FUNCTION_BLOCK FB_ScopeServer
VAR_INPUT
	//sNetId					: STRING	:='';	
    bExternalTriggerEvent	: BOOL 	:= FALSE; //Rising edge start recording, falling edge stop and save
	sConfigFile				: STRING; //.tcscopex
	sSaveFile				: STRING; //.svdx
END_VAR
//VAR_OUTPUT
VAR
    bBusy					: BOOL 		:= FALSE;
    bError					: BOOL 		:= FALSE;
    nErrorId				: UDINT 	:= 0;	
END_VAR
VAR

    bDone					: BOOL 		:= FALSE;	

    fbScopeServerControl	: FB_ScopeServerControl;
    eReqState				: E_ScopeServerState := SCOPE_SERVER_IDLE;
	
    eState					: (IDLE,RECORDING,SAVING,DISCONNECTING,ERROR,RESETING);
END_VAR

CASE eState OF
	IDLE:
		bBusy	:=FALSE;
		IF bExternalTriggerEvent THEN
			bBusy			:= TRUE;
	    	eReqState 		:= SCOPE_SERVER_START;
	    	eState 			:= RECORDING;	
		END_IF
	
	RECORDING:	
		IF fbScopeServerControl.bDone THEN
	    	IF NOT bExternalTriggerEvent THEN
	    	    eReqState 		:= SCOPE_SERVER_SAVE;
	    	    eState 			:= SAVING;
	    	END_IF
		ELSIF fbScopeServerControl.bError THEN
			eState	:=ERROR;		
		END_IF
		
	SAVING:
	    IF fbScopeServerControl.bDone THEN
	        eReqState 		:= SCOPE_SERVER_DISCONNECT;
			eState			:= DISCONNECTING;
		ELSIF fbScopeServerControl.bError THEN
			eState	:=ERROR;		
		END_IF
		
	DISCONNECTING:
		IF fbScopeServerControl.bDone THEN
	       eState := IDLE;
		ELSIF fbScopeServerControl.bError THEN
			eState	:=ERROR;				   
	    END_IF		
		
	ERROR:
		bBusy			:= FALSE;
		IF NOT bExternalTriggerEvent THEN
			bBusy			:= TRUE;
			eReqState 		:= SCOPE_SERVER_RESET;
			eState			:= DISCONNECTING;
		END_IF
		
	RESETING:
		IF fbScopeServerControl.bDone OR fbScopeServerControl.bError THEN
	       	eReqState 		:= SCOPE_SERVER_IDLE;
			eState			:= IDLE; 
	    END_IF		
		
END_CASE


fbScopeServerControl( sNetId		:= '',
                      eReqState		:= eReqState,
                      sConfigFile	:= sConfigFile,
                      sSaveFile		:= sSaveFile,
                      tTimeout		:= T#10S,
                      bBusy			=>,
                      bDone			=>bDone,
                      bError		=>bError,
                      nErrorId		=>nErrorId);

END_FUNCTION_BLOCK

(* stored: Version 1.1.0.1
   POU FB_ScopeServer: Id {2a934d08-2426-4f56-8017-5dfe1fd880a6}, SpecialFunc None *)
